(* Logix 5000 project; controller NorthLineDepalletizerPLC vendor 1 type 14 code 106 rev 33.11; software revision 33.00; part 4 of 4 *)
(* tags used below, declared in another part *)
   ActiveUserFrame : DINT;   // Currently Active Pallet
   AirPressure : ALIAS FOR YRC1000_Rbt_Ctlr:I.Data[1].4;
   Alarm : ALIAS FOR YRC1000_Rbt_Ctlr:I.Data[8].3;
   AlarmReset : ALIAS FOR YRC1000_Rbt_Ctlr:O.Data[0].3;
   Blue1 : BOOL;
   Blue2 : BOOL;
   CallMaster : ALIAS FOR YRC1000_Rbt_Ctlr:O.Data[0].2;
   CameraJobName : STRING;
   ChangingJob : BOOL;
   delay_LeftConveyorOff : TIMER;
   delay_LeftConveyorOffLong : TIMER;
   delay_LeftConveyorOn : TIMER;
   delay_LeftPalletOff : TIMER;
   delay_LeftPalletOn : TIMER;
   delay_RightConveyorOff : TIMER;
   delay_RightConveyorOffLong : TIMER;
   delay_RightConveyorOn : TIMER;
   delay_RightPalletOff : TIMER;
   delay_RightPalletOn : TIMER;
   DoorEntryRequested : ALIAS FOR YRC1000_Rbt_Ctlr:O.Data[5].3;
   DoorLatchRelayPower : ALIAS FOR YRC1000_Rbt_Ctlr:O.Data[2].3;
   DoorRequestAccess : ALIAS FOR YRC1000_Rbt_Ctlr:I.Data[1].0;
   err_CameraFailed : BOOL;
   err_HeightCheckInconsistent : ALIAS FOR YRC1000_Rbt_Ctlr:O.Data[6].3;
   err_RobotPickupFailed : ALIAS FOR YRC1000_Rbt_Ctlr:I.Data[10].3;
   ExternalHold : ALIAS FOR YRC1000_Rbt_Ctlr:O.Data[0].1;
   ExternalServoOn : ALIAS FOR YRC1000_Rbt_Ctlr:O.Data[0].4;
   ExternalStart : ALIAS FOR YRC1000_Rbt_Ctlr:O.Data[0].0;
   GoHome : ALIAS FOR YRC1000_Rbt_Ctlr:O.Data[6].6;
   GoodToPick : ALIAS FOR YRC1000_Rbt_Ctlr:O.Data[8].0;
   GoToToolChange : ALIAS FOR YRC1000_Rbt_Ctlr:O.Data[6].0;
   Green1 : BOOL;
   Green2 : BOOL;
   Gripper_HoldingPart : ALIAS FOR YRC1000_Rbt_Ctlr:O.Data[4].7;
   HMI_GoHome : BOOL;
   HMI_Reset : BOOL;
   HMI_Start : BOOL;
   HMI_Stop : BOOL;
   HMI_Stop_Now : BOOL;
   IFM_Device_Disconnected : BOOL;
   InRemote : ALIAS FOR YRC1000_Rbt_Ctlr:I.Data[8].5;
   InToolChange : ALIAS FOR YRC1000_Rbt_Ctlr:I.Data[10].5;
   JobNamePrefix : STRING;
   LeftConveyorPresent : ALIAS FOR YRC1000_Rbt_Ctlr:O.Data[7].6;
   LeftConveyorSensor : ALIAS FOR YRC1000_Rbt_Ctlr:I.Data[1].5;
   LeftIndicator_Green : ALIAS FOR YRC1000_Rbt_Ctlr:O.Data[1].6;
   LeftIndicator_Yellow : ALIAS FOR YRC1000_Rbt_Ctlr:O.Data[1].7;
   LeftPalletComplete : ALIAS FOR YRC1000_Rbt_Ctlr:O.Data[4].0;
   LeftPalletPresent : ALIAS FOR YRC1000_Rbt_Ctlr:O.Data[7].1;
   LeftPalletSensor : ALIAS FOR YRC1000_Rbt_Ctlr:I.Data[1].2;
   LeftPalletWillBeNew : BOOL;
   msg_Write_ActiveUserFrame : MESSAGE;
   msg_Write_CoilType : MESSAGE;
   msg_Write_ConveyorBeforePlace : MESSAGE;
   msg_Write_PartCount : MESSAGE;
   NewPallet : ALIAS FOR YRC1000_Rbt_Ctlr:O.Data[5].2;
   ons_AddPartToQueue : BOOL;
   ons_CallMaster : BOOL;
   ons_LatchStart : BOOL;
   PalletStarted : ALIAS FOR YRC1000_Rbt_Ctlr:I.Data[10].2;
   PalletTooTall : ALIAS FOR YRC1000_Rbt_Ctlr:I.Data[9].6;
   PartLength : DINT;
   PartLength_Current : DINT;   // 17" = 432 mm 30" = 762 mm 41" = 1041 mm
   PartNum : DINT;
   PartNum_Current : DINT;
   PartNumber : STRING;
   PartNumber_Current : STRING;
   PartRows : DINT;
   PartRows_Current : DINT;
   PartThickness : REAL;
   PartThickness_Current : REAL;   // 2r = 34.1 - 34.8 mm 3r = 51.1 - 51.8 mm 4r = 68.2 - 68.9 mm
   PartWidth : DINT;
   PartWidth_Current : DINT;   // 14" = 356 mm 16" = 406 mm 20" = 508 mm 22" = 559 mm 24" = 610 mm 28" = 711 mm 32" = 813 mm
   patternToPickup : REAL;   // Distance from provided pick position to actual pick position on single-stack A-coils
   QuadStack : ALIAS FOR YRC1000_Rbt_Ctlr:O.Data[4].3;
   recovery_CameraFailed : BOOL;
   recovery_HeightCheckFailed : BOOL;
   recovery_PalletTooTall : BOOL;
   recovery_PickupFailed : BOOL;
   Reset : ALIAS FOR YRC1000_Rbt_Ctlr:I.Data[1].1;
   RightConveyorPresent : ALIAS FOR YRC1000_Rbt_Ctlr:O.Data[7].7;
   RightConveyorSensor : ALIAS FOR YRC1000_Rbt_Ctlr:I.Data[1].6;
   RightIndicator_Green : ALIAS FOR YRC1000_Rbt_Ctlr:O.Data[2].0;
   RightIndicator_Yellow : ALIAS FOR YRC1000_Rbt_Ctlr:O.Data[2].1;
   RightPalletComplete : ALIAS FOR YRC1000_Rbt_Ctlr:O.Data[4].1;
   RightPalletPresent : ALIAS FOR YRC1000_Rbt_Ctlr:O.Data[7].2;
   RightPalletSensor : ALIAS FOR YRC1000_Rbt_Ctlr:I.Data[1].3;
   RightPalletWillBeNew : BOOL;
   RobotExternalEStop : ALIAS FOR YRC1000_Rbt_Ctlr:I.Data[4].1;
   RobotRequestStop : ALIAS FOR YRC1000_Rbt_Ctlr:O.Data[5].4;
   RobotTeachPendantEStop : ALIAS FOR YRC1000_Rbt_Ctlr:I.Data[4].2;
   RobotWentHome : ALIAS FOR YRC1000_Rbt_Ctlr:I.Data[9].5;
   Running : ALIAS FOR YRC1000_Rbt_Ctlr:I.Data[8].0;
   SafetyCircuitBroken : ALIAS FOR YRC1000_Rbt_Ctlr:I.Data[4].0;
   SafetyConfig1 : ALIAS FOR YRC1000_Rbt_Ctlr:O.Data[2].5;
   SafetyConfig2 : ALIAS FOR YRC1000_Rbt_Ctlr:O.Data[2].6;
   SafetyConfig3 : ALIAS FOR YRC1000_Rbt_Ctlr:O.Data[2].7;
   SafetyRelayReset : ALIAS FOR YRC1000_Rbt_Ctlr:O.Data[2].4;
   SelectedJobID : DINT;
   ServoOn : ALIAS FOR YRC1000_Rbt_Ctlr:I.Data[8].1;
   SingleStack : ALIAS FOR YRC1000_Rbt_Ctlr:O.Data[4].2;
   StackLight_Blue : ALIAS FOR YRC1000_Rbt_Ctlr:O.Data[1].3;
   StackLight_Green : ALIAS FOR YRC1000_Rbt_Ctlr:O.Data[1].5;
   StackLight_Red : ALIAS FOR YRC1000_Rbt_Ctlr:O.Data[1].2;
   StackLight_Yellow : ALIAS FOR YRC1000_Rbt_Ctlr:O.Data[1].4;
   timer_CallMaster : TIMER;
   timer_GreenFlashOff : TIMER;
   timer_GreenFlashOn : TIMER;
   timer_HMI_Reset : TIMER;
   timer_HMI_Start : TIMER;
   timer_HMI_Stop : TIMER;
   timer_LeftFlashOff : TIMER;
   timer_LeftFlashOn : TIMER;
   timer_RightFlashOff : TIMER;
   timer_RightFlashOn : TIMER;
   TopOfMaster : ALIAS FOR YRC1000_Rbt_Ctlr:I.Data[8].2;
   Write_ActiveUserFrame : BOOL;
   write_ActiveUserFrame_L : BOOL;
   Write_ActiveUserFrame_R : BOOL;
   Write_CoilType : BOOL;
   Write_ConveyorPositions : BOOL;
   Write_PartCount : BOOL;
(* Motoman, continued *)

ROUTINE Pallet_StackLight_DoorLatch   (* ladder *)
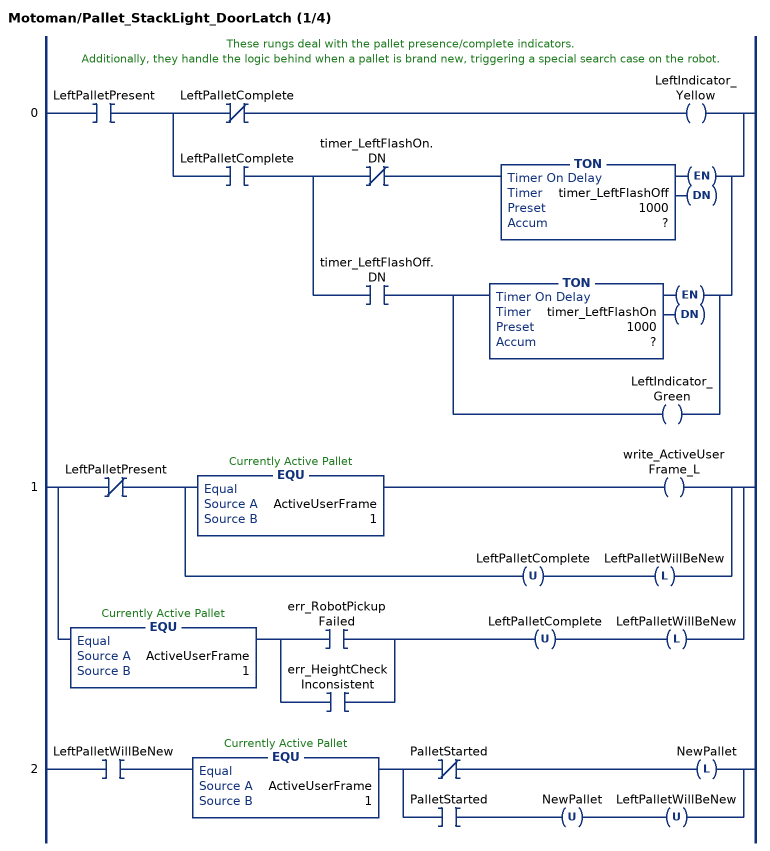
   // These rungs deal with the pallet presence/complete indicators.
   // Additionally, they handle the logic behind when a pallet is brand new, triggering a special search case on the robot.
   0: XIC(LeftPalletPresent)[XIO(LeftPalletComplete) OTE(LeftIndicator_Yellow) ,XIC(LeftPalletComplete) [XIO(timer_LeftFlashOn.DN) TON(timer_LeftFlashOff,?,?) ,XIC(timer_LeftFlashOff.DN) [TON(timer_LeftFlashOn,?,?) ,OTE(LeftIndicator_Green) ] ] ];
   1: [XIO(LeftPalletPresent) [EQU(ActiveUserFrame,1) OTE(write_ActiveUserFrame_L) ,OTU(LeftPalletComplete) OTL(LeftPalletWillBeNew) ] ,EQU(ActiveUserFrame,1) [XIC(err_RobotPickupFailed) ,XIC(err_HeightCheckInconsistent) ] OTU(LeftPalletComplete) OTL(LeftPalletWillBeNew) ];
   2: XIC(LeftPalletWillBeNew)EQU(ActiveUserFrame,1)[XIO(PalletStarted) OTL(NewPallet) ,XIC(PalletStarted) OTU(NewPallet) OTU(LeftPalletWillBeNew) ];
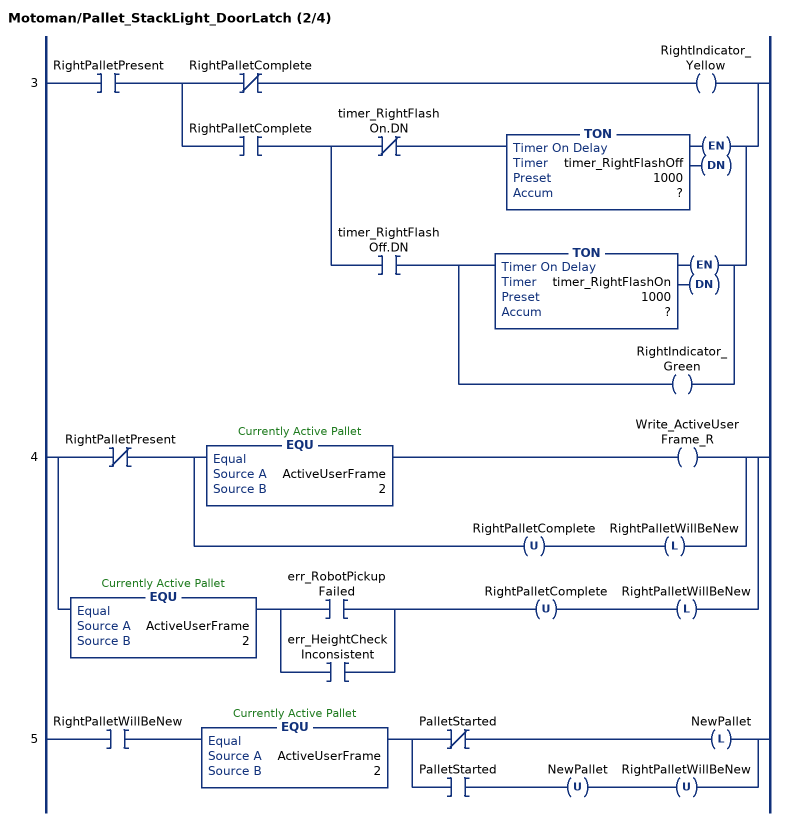
   3: XIC(RightPalletPresent)[XIO(RightPalletComplete) OTE(RightIndicator_Yellow) ,XIC(RightPalletComplete) [XIO(timer_RightFlashOn.DN) TON(timer_RightFlashOff,?,?) ,XIC(timer_RightFlashOff.DN) [TON(timer_RightFlashOn,?,?) ,OTE(RightIndicator_Green) ] ] ];
   4: [XIO(RightPalletPresent) [EQU(ActiveUserFrame,2) OTE(Write_ActiveUserFrame_R) ,OTU(RightPalletComplete) OTL(RightPalletWillBeNew) ] ,EQU(ActiveUserFrame,2) [XIC(err_RobotPickupFailed) ,XIC(err_HeightCheckInconsistent) ] OTU(RightPalletComplete) OTL(RightPalletWillBeNew) ];
   5: XIC(RightPalletWillBeNew)EQU(ActiveUserFrame,2)[XIO(PalletStarted) OTL(NewPallet) ,XIC(PalletStarted) OTU(NewPallet) OTU(RightPalletWillBeNew) ];
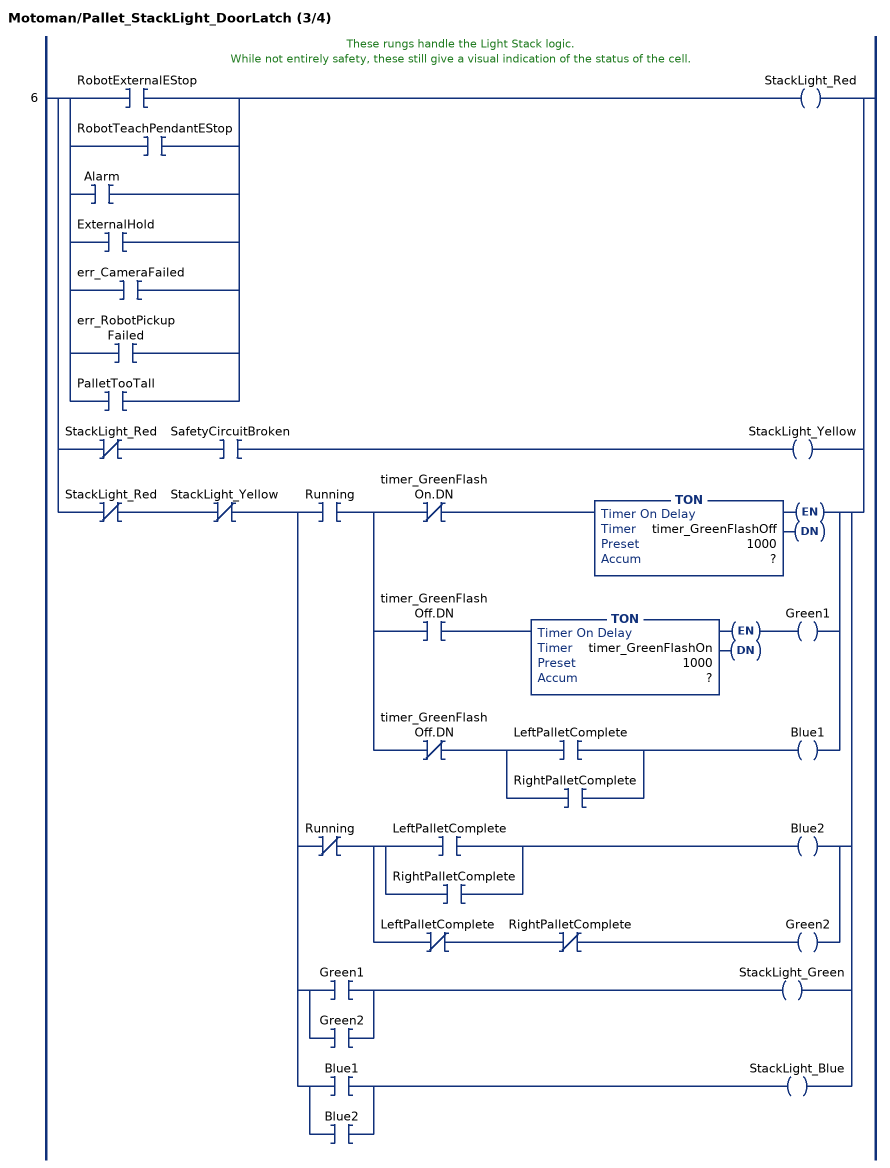
   // These rungs handle the Light Stack logic.
   // While not entirely safety, these still give a visual indication of the status of the cell.
   6: [[XIC(RobotExternalEStop) ,XIC(RobotTeachPendantEStop) ,XIC(Alarm) ,XIC(ExternalHold) ,XIC(err_CameraFailed) ,XIC(err_RobotPickupFailed) ,XIC(PalletTooTall) ] OTE(StackLight_Red) ,XIO(StackLight_Red) XIC(SafetyCircuitBroken) OTE(StackLight_Yellow) ,XIO(StackLight_Red) XIO(StackLight_Yellow) [[XIC(Running) [XIO(timer_GreenFlashOn.DN) TON(timer_GreenFlashOff,?,?) ,XIC(timer_GreenFlashOff.DN) TON(timer_GreenFlashOn,?,?) OTE(Green1) ,XIO(timer_GreenFlashOff.DN) [XIC(LeftPalletComplete) ,XIC(RightPalletComplete) ] OTE(Blue1) ] ,XIO(Running) [[XIC(LeftPalletComplete) ,XIC(RightPalletComplete) ] OTE(Blue2) ,XIO(LeftPalletComplete) XIO(RightPalletComplete) OTE(Green2) ] ] ,[XIC(Green1) ,XIC(Green2) ] OTE(StackLight_Green) ,[XIC(Blue1) ,XIC(Blue2) ] OTE(StackLight_Blue) ] ];
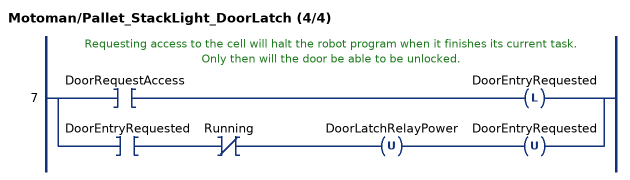
   // Requesting access to the cell will halt the robot program when it finishes its current task.
   // Only then will the door be able to be unlocked.
   7: [XIC(DoorRequestAccess) OTL(DoorEntryRequested) ,XIC(DoorEntryRequested) XIO(Running) OTU(DoorLatchRelayPower) OTU(DoorEntryRequested) ];
END_ROUTINE

ROUTINE PartChange   (* ladder *)
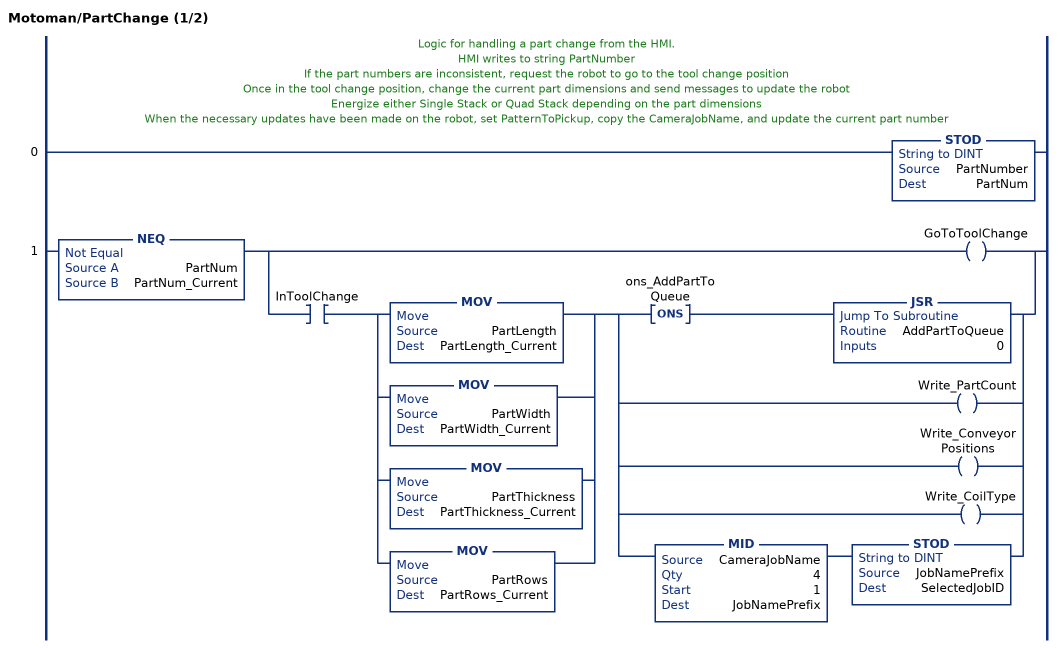
   // Logic for handling a part change from the HMI.
   // HMI writes to string PartNumber
   // If the part numbers are inconsistent, request the robot to go to the tool change position
   // Once in the tool change position, change the current part dimensions and send messages to update the robot
   // Energize either Single Stack or Quad Stack depending on the part dimensions
   // When the necessary updates have been made on the robot, set PatternToPickup, copy the CameraJobName, and update the current part number
   0: STOD(PartNumber,PartNum);
   1: NEQ(PartNum,PartNum_Current)[OTE(GoToToolChange) ,XIC(InToolChange) [MOV(PartLength,PartLength_Current) ,MOV(PartWidth,PartWidth_Current) ,MOV(PartThickness,PartThickness_Current) ,MOV(PartRows,PartRows_Current) ] [ONS(ons_AddPartToQueue) JSR(AddPartToQueue,0) ,OTE(Write_PartCount) ,OTE(Write_ConveyorPositions) ,OTE(Write_CoilType) ,MID(CameraJobName,4,1,JobNamePrefix) STOD(JobNamePrefix,SelectedJobID) ] ];
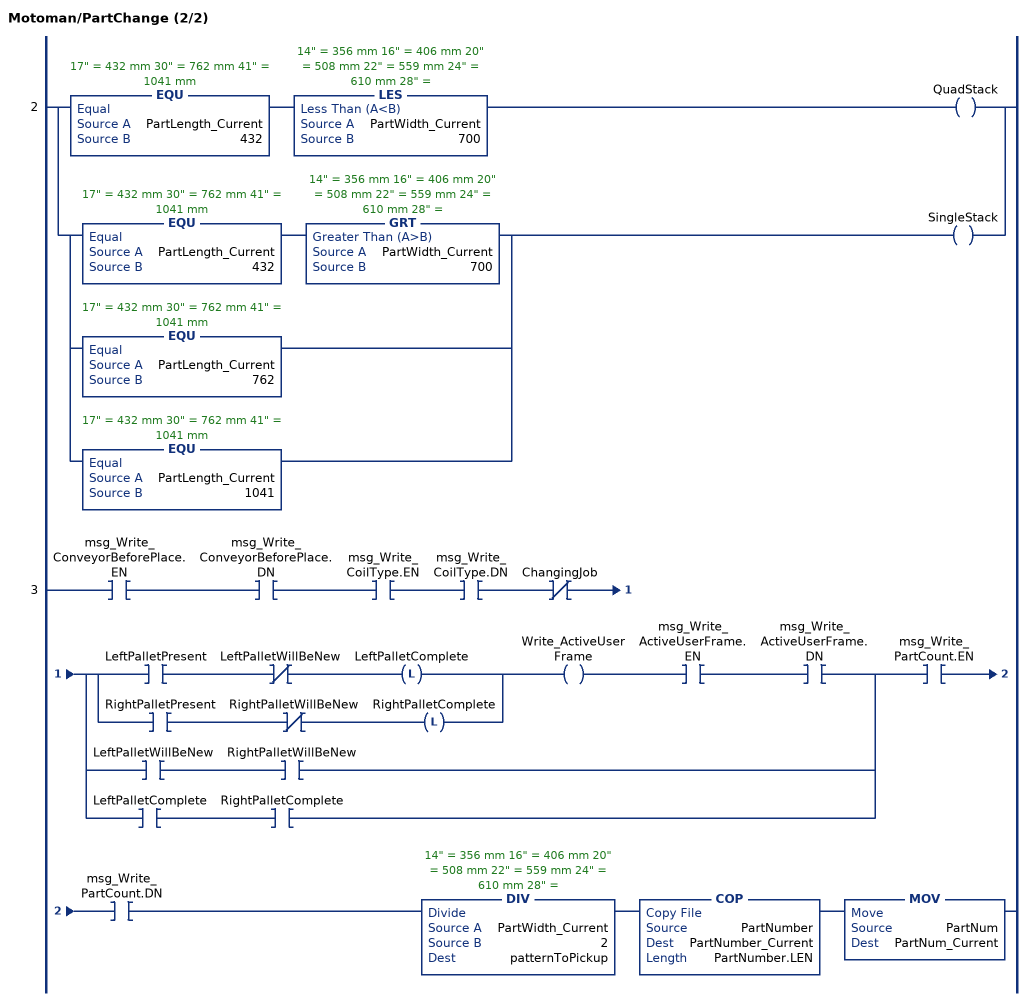
   2: [EQU(PartLength_Current,432) LES(PartWidth_Current,700) OTE(QuadStack) ,[EQU(PartLength_Current,432) GRT(PartWidth_Current,700) ,EQU(PartLength_Current,762) ,EQU(PartLength_Current,1041) ] OTE(SingleStack) ];
   3: XIC(msg_Write_ConveyorBeforePlace.EN)XIC(msg_Write_ConveyorBeforePlace.DN)XIC(msg_Write_CoilType.EN)XIC(msg_Write_CoilType.DN)XIO(ChangingJob)[[XIC(LeftPalletPresent) XIO(LeftPalletWillBeNew) OTL(LeftPalletComplete) ,XIC(RightPalletPresent) XIO(RightPalletWillBeNew) OTL(RightPalletComplete) ] OTE(Write_ActiveUserFrame) XIC(msg_Write_ActiveUserFrame.EN) XIC(msg_Write_ActiveUserFrame.DN) ,[XIC(LeftPalletWillBeNew) XIC(RightPalletWillBeNew) ,XIC(LeftPalletComplete) XIC(RightPalletComplete) ] ]XIC(msg_Write_PartCount.EN)XIC(msg_Write_PartCount.DN)DIV(PartWidth_Current,2,patternToPickup)COP(PartNumber,PartNumber_Current,PartNumber.LEN)MOV(PartNum,PartNum_Current);
END_ROUTINE

ROUTINE SafeyScannerZones   (* ladder *)
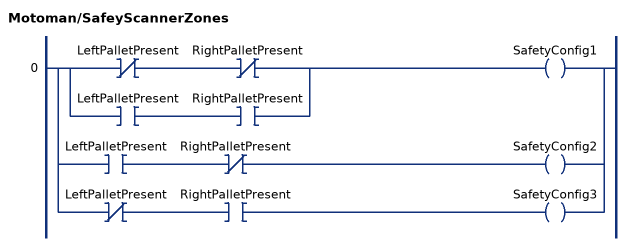
   0: [[XIO(LeftPalletPresent) XIO(RightPalletPresent) ,XIC(LeftPalletPresent) XIC(RightPalletPresent) ] OTE(SafetyConfig1) ,XIC(LeftPalletPresent) XIO(RightPalletPresent) OTE(SafetyConfig2) ,XIO(LeftPalletPresent) XIC(RightPalletPresent) OTE(SafetyConfig3) ];
END_ROUTINE

ROUTINE SensorDelays   (* ladder *)
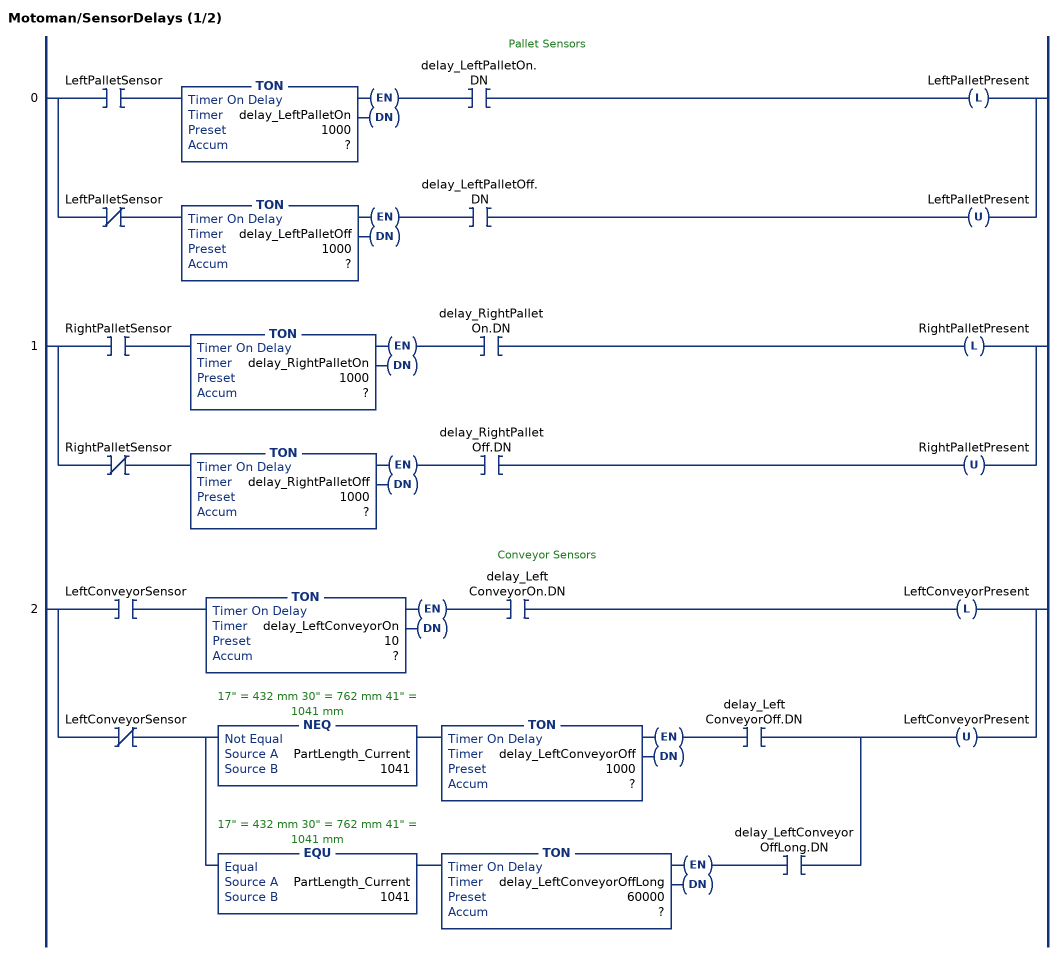
   // Pallet Sensors
   0: [XIC(LeftPalletSensor) TON(delay_LeftPalletOn,?,?) XIC(delay_LeftPalletOn.DN) OTL(LeftPalletPresent) ,XIO(LeftPalletSensor) TON(delay_LeftPalletOff,?,?) XIC(delay_LeftPalletOff.DN) OTU(LeftPalletPresent) ];
   1: [XIC(RightPalletSensor) TON(delay_RightPalletOn,?,?) XIC(delay_RightPalletOn.DN) OTL(RightPalletPresent) ,XIO(RightPalletSensor) TON(delay_RightPalletOff,?,?) XIC(delay_RightPalletOff.DN) OTU(RightPalletPresent) ];
   // Conveyor Sensors
   2: [XIC(LeftConveyorSensor) TON(delay_LeftConveyorOn,?,?) XIC(delay_LeftConveyorOn.DN) OTL(LeftConveyorPresent) ,XIO(LeftConveyorSensor) [NEQ(PartLength_Current,1041) TON(delay_LeftConveyorOff,?,?) XIC(delay_LeftConveyorOff.DN) ,EQU(PartLength_Current,1041) TON(delay_LeftConveyorOffLong,?,?) XIC(delay_LeftConveyorOffLong.DN) ] OTU(LeftConveyorPresent) ];
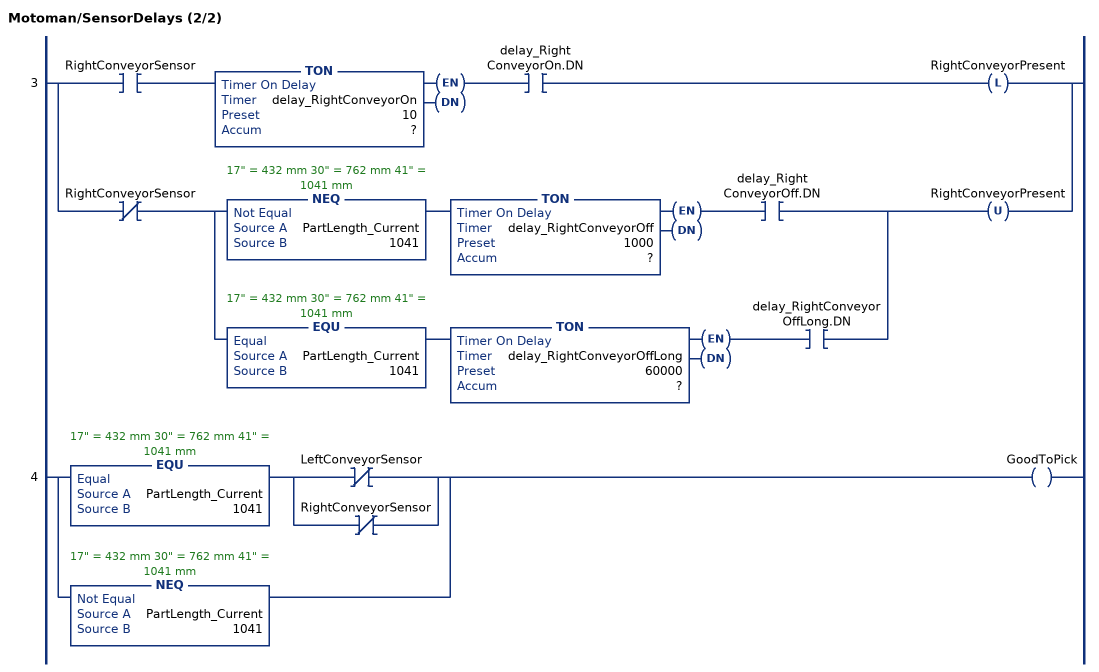
   3: [XIC(RightConveyorSensor) TON(delay_RightConveyorOn,?,?) XIC(delay_RightConveyorOn.DN) OTL(RightConveyorPresent) ,XIO(RightConveyorSensor) [NEQ(PartLength_Current,1041) TON(delay_RightConveyorOff,?,?) XIC(delay_RightConveyorOff.DN) ,EQU(PartLength_Current,1041) TON(delay_RightConveyorOffLong,?,?) XIC(delay_RightConveyorOffLong.DN) ] OTU(RightConveyorPresent) ];
   4: [EQU(PartLength_Current,1041) [XIO(LeftConveyorSensor) ,XIO(RightConveyorSensor) ] ,NEQ(PartLength_Current,1041) ]OTE(GoodToPick);
END_ROUTINE

ROUTINE Start_Stop_Reset   (* ladder *)
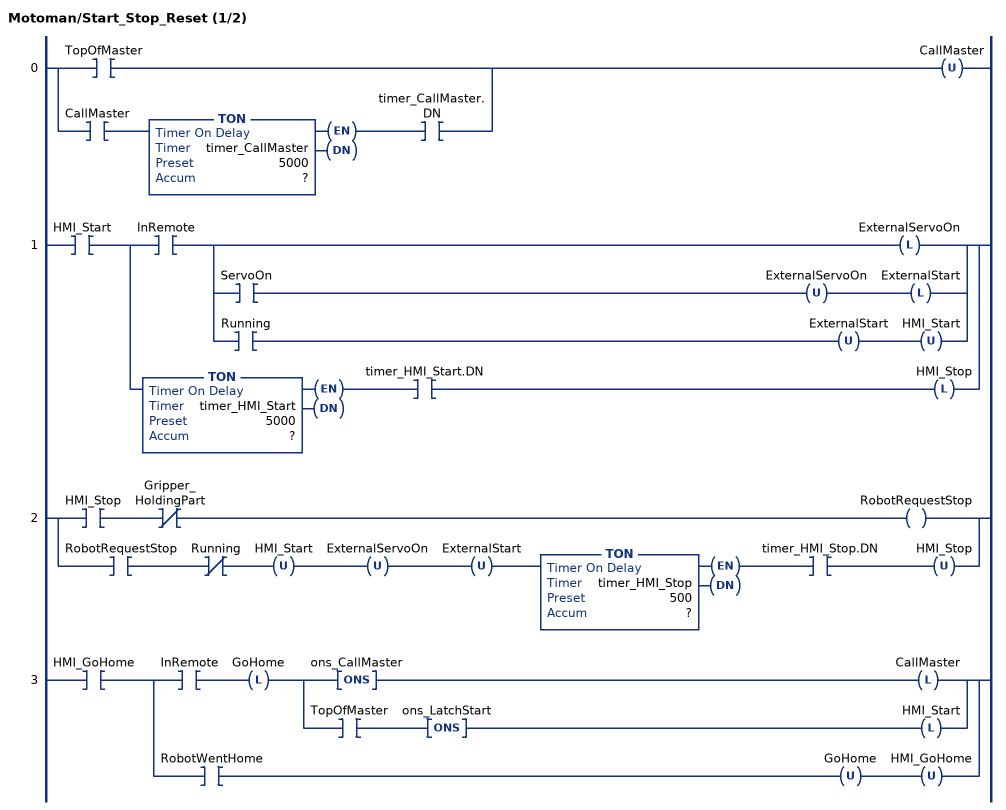
   0: [XIC(TopOfMaster) ,XIC(CallMaster) TON(timer_CallMaster,?,?) XIC(timer_CallMaster.DN) ]OTU(CallMaster);
   1: XIC(HMI_Start)[XIC(InRemote) [OTL(ExternalServoOn) ,XIC(ServoOn) OTU(ExternalServoOn) OTL(ExternalStart) ,XIC(Running) OTU(ExternalStart) OTU(HMI_Start) ] ,TON(timer_HMI_Start,?,?) XIC(timer_HMI_Start.DN) OTL(HMI_Stop) ];
   2: [XIC(HMI_Stop) XIO(Gripper_HoldingPart) OTE(RobotRequestStop) ,XIC(RobotRequestStop) XIO(Running) OTU(HMI_Start) OTU(ExternalServoOn) OTU(ExternalStart) TON(timer_HMI_Stop,?,?) XIC(timer_HMI_Stop.DN) OTU(HMI_Stop) ];
   3: XIC(HMI_GoHome)[XIC(InRemote) OTL(GoHome) [ONS(ons_CallMaster) OTL(CallMaster) ,XIC(TopOfMaster) ONS(ons_LatchStart) OTL(HMI_Start) ] ,XIC(RobotWentHome) OTU(GoHome) OTU(HMI_GoHome) ];
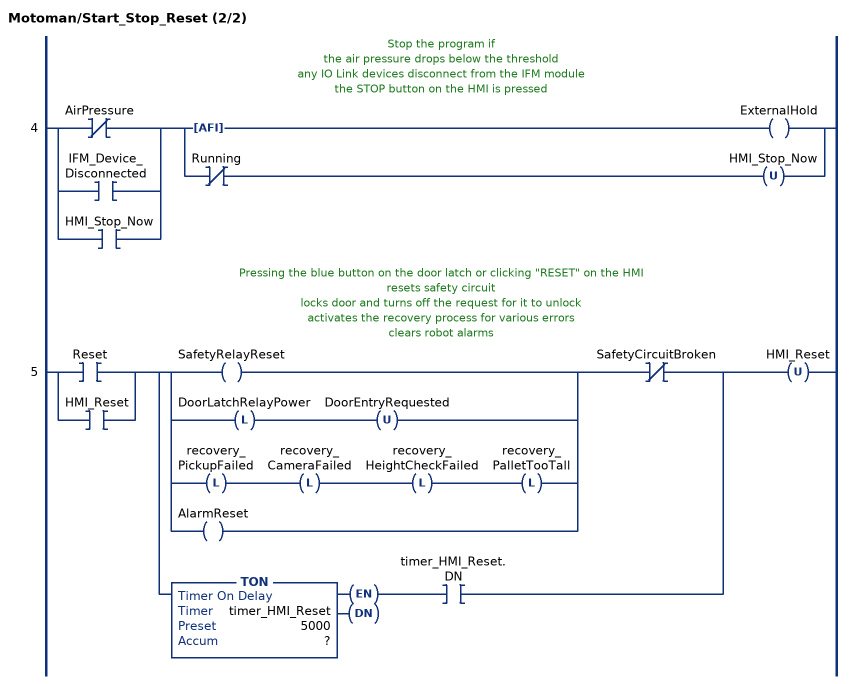
   // Stop the program if
   //      the air pressure drops below the threshold
   //      any IO Link devices disconnect from the IFM module
   //      the STOP button on the HMI is pressed
   4: [XIO(AirPressure) ,XIC(IFM_Device_Disconnected) ,XIC(HMI_Stop_Now) ][AFI() OTE(ExternalHold) ,XIO(Running) OTU(HMI_Stop_Now) ];
   // Pressing the blue button on the door latch or clicking "RESET" on the HMI
   //      resets safety circuit
   //      locks door and turns off the request for it to unlock
   //      activates the recovery process for various errors
   //      clears robot alarms
   5: [XIC(Reset) ,XIC(HMI_Reset) ][[OTE(SafetyRelayReset) ,OTL(DoorLatchRelayPower) OTU(DoorEntryRequested) ,OTL(recovery_PickupFailed) OTL(recovery_CameraFailed) OTL(recovery_HeightCheckFailed) OTL(recovery_PalletTooTall) ,OTE(AlarmReset) ] XIO(SafetyCircuitBroken) ,TON(timer_HMI_Reset,?,?) XIC(timer_HMI_Reset.DN) ]OTU(HMI_Reset);
END_ROUTINE
END_PROGRAM
